ABB RAPID module: A098_DataTask_Rob.mod

MODULE A098_DataTask_Rob
    !***********************************************************************************
    !
    ! ETH Zurich / NCCR Digital Fabrication
    ! HIB C51 / Stefano-Franscini-Platz 1
    ! CH-8093 Zurich
    !
    !***********************************************************************************
    !
    ! PROJECT     :  A098 Fall_Demo_2025
    !
    ! FUNCTION    :  Includ all Task Data's for Project
    !
    ! AUTHOR      :  Philippe Fleischmann
    !
    ! EMAIL       :  fleischmann@arch.ethz.ch
    !
    ! HISTORY     :  2025.10.31
    !
    ! Copyright   :  ETH Zurich (CH) 2022
    !
    !***********************************************************************************

    !************************************************
    ! Declaration :     bool
    !************************************************
    !
    TASK PERS bool b_A098_MyBool:=FALSE;

    !************************************************
    ! Declaration :     num
    !************************************************
    !
    TASK PERS num n_A098_MyNum:=0;

    !************************************************
    ! Declaration :     string
    !************************************************
    !
    TASK PERS string st_A098_MyString:="";

    !************************************************
    ! Declaration :     tooldata
    !************************************************
    !
    TASK PERS tooldata t_A098_gripper_beams_falld:=[TRUE,[[0.951252,0.594269,204.442],[1,0,0,0]],[10,[0,0,0],[1,0,0,0],0,0,0]];
    TASK PERS tooldata t_A098_gripper_1:=[TRUE,[[0,0,300],[1,0,0,0]],[40,[0,0,332],[1,0,0,0],0,0,0]];

    !************************************************
    ! Declaration :     wobjdata
    !************************************************
    !
	TASK PERS wobjdata ob_A098_pick_up_station:=[FALSE,TRUE,"",[[12608.8,1065.47,988.007],[6.55418E-06,-8.44528E-05,-0.000586165,-1]],[[0,0,0],[1,0,0,0]]];
	TASK PERS wobjdata ob_A098_cnc_left_corner:=[FALSE,TRUE,"",[[12608.8,1065.47,988.007],[6.55418E-06,-8.44528E-05,-0.000586165,-1]],[[0,0,0],[1,0,0,0]]];
	TASK PERS wobjdata ob_A098_assembly_table:=[FALSE,TRUE,"",[[8717.23,6132,745.795],[0.999989,-0.00321826,0.00278036,0.00215958]],[[0,0,0],[1,0,0,0]]];

    !************************************************
    ! Declaration :     jointtarget
    !************************************************
    !
    TASK PERS jointtarget jp_A098_MyJointtarget:=[[0,0,0,0,0,0],[9E9,9E9,9E9,9E9,9E9,9E9]];

    !************************************************
    ! Declaration :     robtarget
    !************************************************
    !
    TASK PERS robtarget p_A098_MyRobtarget:=[[0,0,0],[1,0,0,0],[0,0,0,0],[9E9,9E9,9E9,9E9,9E9,9E9]];

    !************************************************
    ! Declaration :     speeddata
    !************************************************
    !
    TASK PERS speeddata v_A098_MySpeed:=[0,0,0,0];
    TASK PERS tooldata t_A098_gripper_2:=[TRUE,[[0,0,300],[1,0,0,0]],[10,[0,0,150],[1,0,0,0],0,0,0]];
    TASK PERS tooldata t_A098_GoldenGripper:=[TRUE,[[-0.0455761,-1.29732,400.807],[1,0,0,0]],[50,[-0.0455761,-1.29732,300.807],[1,0,0,0],0,0,0]];
    TASK PERS wobjdata bps_fd:=[FALSE,TRUE,"",[[10999.9,5290.72,474.41],[0.00226011,-0.000813826,-0.371826,0.928299]],[[0,0,0],[1,0,0,0]]];
    TASK PERS wobjdata ob_A098_bps:=[FALSE,TRUE,"",[[11072.5,5287.75,472.392],[0.000604694,0.00284125,0.926429,0.376459]],[[0,0,0],[1,0,0,0]]];
ENDMODULE
